// TIA Portal V18 program export: 5 tag tables, 0 data types, 0 data blocks, 6 code blocks (in call order from the OBs), 5 instance data blocks

VAR_GLOBAL   // PLC tag table "Default tag table"
   System_Byte AT %MB1 : Byte;
   FirstScan AT %M1.0 : Bool;
   DiagStatusUpdate AT %M1.1 : Bool;
   AlwaysTRUE AT %M1.2 : Bool;
   AlwaysFALSE AT %M1.3 : Bool;
   Clock_Byte AT %MB0 : Byte;
   Clock_10Hz AT %M0.0 : Bool;
   Clock_5Hz AT %M0.1 : Bool;
   "Clock_2.5Hz" AT %M0.2 : Bool;
   Clock_2Hz AT %M0.3 : Bool;
   "Clock_1.25Hz" AT %M0.4 : Bool;
   Clock_1Hz AT %M0.5 : Bool;
   "Clock_0.625Hz" AT %M0.6 : Bool;
   "Clock_0.5Hz" AT %M0.7 : Bool;
   rozlaczenie_tasmy AT %M100.2 : Bool;
   reset_licznika AT %M100.3 : Bool;
   zatrzymanie_tasmy AT %M101.2 : Bool;
   ilosc_butelek AT %MW10 : Int;
   reset_licznika_zak AT %M101.3 : Bool;
   ilosc_butelek_zak AT %MW16 : Int;
   Wylacznik_bezpieczenstwa AT %M205.0 : Bool;
   "Wlacznik/Wylacznik_glowny" AT %M206.0 : Bool;
   start_przenosik AT %M204.0 : Bool;
   stop_przenosnik AT %M204.1 : Bool;
   przenosnik_tasmowy AT %Q1.4 : Bool;
   wylacznik_przenosnika_tasmowego AT %I1.4 : Bool;
   wylacznik_nalewarki AT %I1.5 : Bool;
   wylacznik_zakrecarki AT %I1.6 : Bool;
   wylacznik_etykieciarki AT %I1.7 : Bool;
   wylacznik_pakowanie AT %I2.0 : Bool;
   samopod_start_zak AT %M102.3 : Bool;
   samopod_start_nal AT %M100.4 : Bool;
   Wlacznik_500ml AT %M207.0 : Bool;
   silownik AT %Q1.5 : Bool;
   sygnalizator_dzwiekowy AT %Q2.2 : Bool;
   robot AT %Q2.3 : Bool;
   lampa_przenosnik AT %Q2.4 : Bool;
   licznik_etykiet AT %MW50 : Int;
   cz_poj_ety AT %M210.0 : Bool;
   reset_licznika_etyk AT %M211.0 : Bool;
   pamiec_smakow AT %M100.5 : Bool;
   smak_zatrzymaj AT %M212.2 : Bool;
   czas_nalewarka AT %MD300 : Time;
   czas_pakowanie AT %MD304 : Time;
   czas_zakrecarka AT %MD308 : Time;
   cz_butelek_pakowanie AT %M230.0 : Bool;
   Tag_1 AT %MW400 : Word;
   licznik_przenosnik AT %MW30 : Int;
   res_licz_przen AT %M350.0 : Bool;
   Tag_4 AT %MD32 : Time;
   Tag_5 AT %M500.0 : Bool;
   res_licz_nalew AT %M350.1 : Bool;
   licznik_nalewarak AT %MW34 : Int;
   Tag_2 AT %M350.2 : Bool;
   Tag_3 AT %MW38 : Word;
   czas_move AT %MD312 : DWord;
   czas_w_int AT %MD316 : UDInt;
   Tag_6 AT %M320.0 : Bool;
   Tag_7 AT %MD321 : Time;
   Tag_8 AT %MD325 : Time;
   Tag_9 AT %MD329 : DInt;
   Tag_10 AT %I90.0 : Bool;
END_VAR

VAR_GLOBAL   // PLC tag table "Etykieciarka"
   start_etykieciarka AT %M102.0 : Bool;
   stop_etykieciarka AT %M102.1 : Bool;
   cz_swiatlowodowy AT %M202.0 : Bool;
   etykieta AT %Q0.6 : Bool;
   tasma_etykieciarka AT %Q0.7 : Bool;
   lampa_sygnalizacyjna_etyk AT %Q1.0 : Bool;
END_VAR

VAR_GLOBAL   // PLC tag table "Nalewarka"
   start_nalewarka AT %M100.0 : Bool;
   stop_nalewarka AT %M100.1 : Bool;
   cz_pojemnosciowy AT %M200.0 : Bool;
   dozy AT %Q0.1 : Bool;
   tasma AT %Q0.0 : Bool;
   lampa AT %Q0.2 : Bool;
   wl_pomarancza AT %M212.0 : Bool;
   pomarancza AT %Q2.5 : Bool;
   wl_truskawka AT %M212.1 : Bool;
   truskawka AT %Q2.6 : Bool;
   cz_poz_napoju AT %M213.0 : Bool;
END_VAR

VAR_GLOBAL   // PLC tag table "Pakowanie"
   start_pakowaie AT %M103.0 : Bool;
   stop_pakowanie AT %M103.1 : Bool;
   cz_pojemnosciowy_pak AT %M203.0 : Bool;
   tasma_pakowanie AT %Q1.2 : Bool;
   lampa_sygnalizacyjna_pak AT %Q1.1 : Bool;
   cz_do_robota AT %Q1.3 : Bool;
END_VAR

VAR_GLOBAL   // PLC tag table "Zakrecarka"
   start_zakrecarka AT %M101.0 : Bool;
   stop_zakrecarka AT %M101.1 : Bool;
   cz_pojemnosciowy_zak AT %M201.0 : Bool;
   tasma_zakrecarka AT %Q0.4 : Bool;
   zakretka AT %Q0.3 : Bool;
   lampa_sygnalizacyjna AT %Q0.5 : Bool;
END_VAR

ORGANIZATION_BLOCK "Main"   // OB1, LAD, ProgramCycle
TITLE = "Main Program Sweep (Cycle)"
{ S7_Optimized_Access := 'TRUE' }
VERSION : 0.1
// stored: AutoNumber true, IsIECCheckEnabled false, SetENOAutomatically false
   VAR_INPUT
      Initial_Call : Bool;   // Initial call of this OB
      Remanence : Bool;   // =True, if remanent data are available
   END_VAR
   VAR_TEMP   // added for the SCL form of the ladder/FBD networks
      _w1 : Bool;
      _w2 : Bool;
      _w3 : Bool;
      _w4 : Bool;
      _w5 : Bool;
   END_VAR
BEGIN

REGION Network 1
   // Linię produkcyjną uruchamiamy poprzez włącznik główny oraz dodatkowo każdy etap produkcji na panelu HMI.
   // Wyłącznik bezpieczeństwa znajduje się w kilku miejscach na linii produkcyjnej.
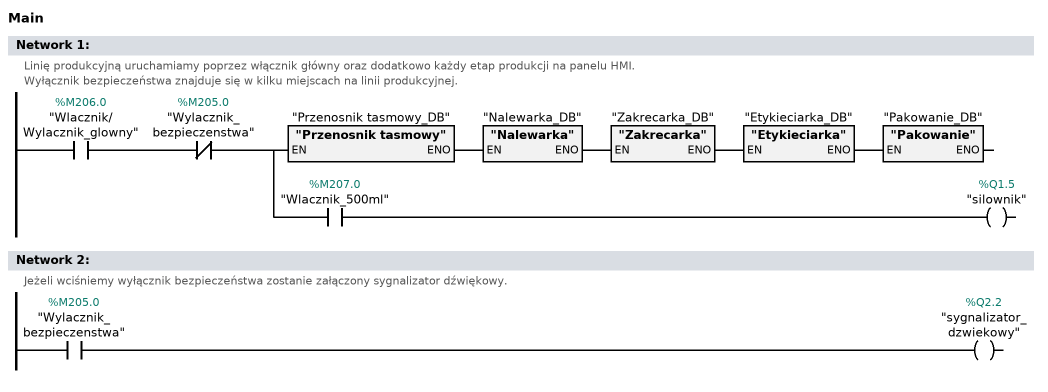
   RUNG wire#powerrail
      Contact( "Wlacznik/Wylacznik_glowny" )
      I_Contact( "Wylacznik_bezpieczenstwa" )
      wire#w1
      "Przenosnik tasmowy_DB"()
      "Nalewarka_DB"()
      "Zakrecarka_DB"()
      "Etykieciarka_DB"()
      "Pakowanie_DB"()
   END_RUNG
   RUNG wire#w1
      Contact( "Wlacznik_500ml" )
      Coil( "silownik" )
   END_RUNG
   // the same network as SCL:
   #_w1 := "Wlacznik/Wylacznik_glowny" AND NOT "Wylacznik_bezpieczenstwa";
   "Przenosnik tasmowy_DB"(EN := #_w1, ENO => #_w2);   // "Przenosnik tasmowy"
   "Nalewarka_DB"(EN := #_w2, ENO => #_w3);   // "Nalewarka"
   "Zakrecarka_DB"(EN := #_w3, ENO => #_w4);   // "Zakrecarka"
   "Etykieciarka_DB"(EN := #_w4, ENO => #_w5);   // "Etykieciarka"
   IF #_w5 THEN
       "Pakowanie_DB"();   // "Pakowanie"
   END_IF;
   "silownik" := #_w1 AND "Wlacznik_500ml";
END_REGION

REGION Network 2
   // Jeżeli wciśniemy wyłącznik bezpieczeństwa zostanie załączony sygnalizator dźwiękowy.
   RUNG wire#powerrail
      Contact( "Wylacznik_bezpieczenstwa" )
      Coil( "sygnalizator_dzwiekowy" )
   END_RUNG
   // the same network as SCL:
   "sygnalizator_dzwiekowy" := "Wylacznik_bezpieczenstwa";
END_REGION
END_ORGANIZATION_BLOCK

FUNCTION_BLOCK "Przenosnik tasmowy"   // FB5, LAD
{ S7_Optimized_Access := 'TRUE' }
VERSION : 0.1
// stored: AutoNumber true, IsIECCheckEnabled false, IsRetainMemResEnabled false, MemoryReserve 100, SetENOAutomatically false, UDAEnableTagReadback false
   VAR_TEMP
      mem0 : Time;
   END_VAR
BEGIN

REGION Network 1
   // Start przenośnika taśmowego.
   // Wyłącznik przenośnika znajduje się fizycznie na linii produkcyjnej. Stop natomiast w panelu HMI.
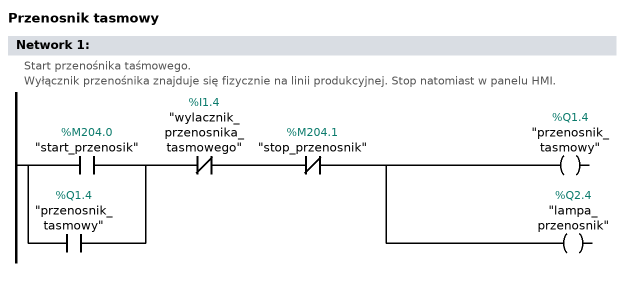
   RUNG wire#powerrail
      Contact( "start_przenosik" )
      wire#w1
      I_Contact( "wylacznik_przenosnika_tasmowego" )
      I_Contact( "stop_przenosnik" )
      wire#w2
      Coil( "przenosnik_tasmowy" )
   END_RUNG
   RUNG wire#powerrail
      Contact( "przenosnik_tasmowy" )
   END_RUNG wire#w1
   RUNG wire#w2
      Coil( "lampa_przenosnik" )
   END_RUNG
   // the same network as SCL:
   "przenosnik_tasmowy" := ("start_przenosik" OR "przenosnik_tasmowy") AND NOT "wylacznik_przenosnika_tasmowego" AND NOT "stop_przenosnik";
   "lampa_przenosnik" := "przenosnik_tasmowy";
END_REGION
END_FUNCTION_BLOCK

FUNCTION_BLOCK "Nalewarka"   // FB1, LAD
{ S7_Optimized_Access := 'TRUE' }
VERSION : 0.1
// stored: AutoNumber true, IsIECCheckEnabled false, IsRetainMemResEnabled false, MemoryReserve 100, SetENOAutomatically false, UDAEnableTagReadback false
   VAR
      czas_nalewarka : Time;
   END_VAR
   VAR_TEMP   // added for the SCL form of the ladder/FBD networks
      _w1 : Bool;
   END_VAR
BEGIN

REGION Network 1
   // Start przenośnika taśmowego i zapalenie się lampy sygnalizacyjnej.
   // Wyłącznik nalewarki znajduje się fizycznie na linii produkcyjnej, w jego skład wchodzi również system ryglowania. Stop natomiast w panelu HMI.
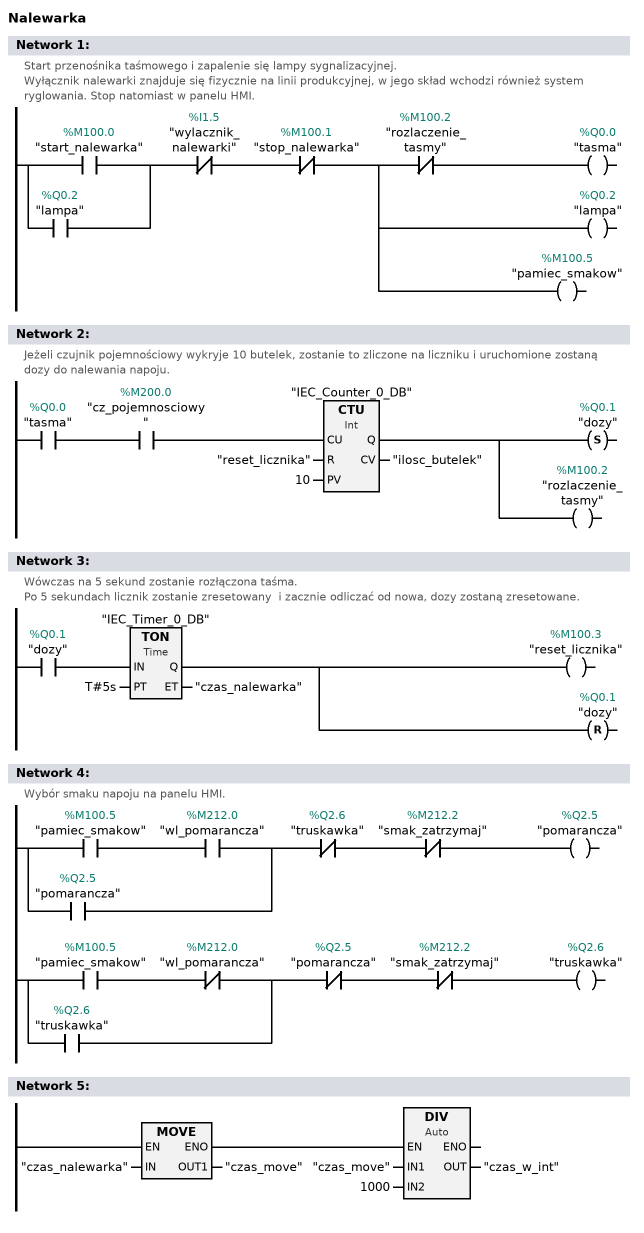
   RUNG wire#powerrail
      Contact( "start_nalewarka" )
      wire#w1
      I_Contact( "wylacznik_nalewarki" )
      I_Contact( "stop_nalewarka" )
      wire#w2
      I_Contact( "rozlaczenie_tasmy" )
      Coil( "tasma" )
   END_RUNG
   RUNG wire#powerrail
      Contact( "lampa" )
   END_RUNG wire#w1
   RUNG wire#w2
      Coil( "lampa" )
   END_RUNG
   RUNG wire#w2
      Coil( "pamiec_smakow" )
   END_RUNG
   // the same network as SCL:
   #_w1 := ("start_nalewarka" OR "lampa") AND NOT "wylacznik_nalewarki" AND NOT "stop_nalewarka";
   "tasma" := #_w1 AND NOT "rozlaczenie_tasmy";
   "lampa" := #_w1;
   "pamiec_smakow" := #_w1;
END_REGION

REGION Network 2
   // Jeżeli czujnik pojemnościowy wykryje 10 butelek, zostanie to zliczone na liczniku i uruchomione zostaną dozy do nalewania napoju.
   RUNG wire#powerrail
      Contact( "tasma" )
      Contact( "cz_pojemnosciowy" )
      { S7_Templates := "value_type := Int" } "IEC_Counter_0_DB".CTU(r := "reset_licznika", pv := 10, cv => "ilosc_butelek")
      wire#w1
      S_Coil( "dozy" )
   END_RUNG
   RUNG wire#w1
      Coil( "rozlaczenie_tasmy" )
   END_RUNG
   // the same network as SCL:
   "IEC_Counter_0_DB".CTU(CU := "tasma" AND "cz_pojemnosciowy",
                          R := "reset_licznika",
                          PV := 10,
                          CV => "ilosc_butelek");
   IF "IEC_Counter_0_DB".Q THEN "dozy" := TRUE; END_IF;
   "rozlaczenie_tasmy" := "IEC_Counter_0_DB".Q;
END_REGION

REGION Network 3
   // Wówczas na 5 sekund zostanie rozłączona taśma.
   // Po 5 sekundach licznik zostanie zresetowany  i zacznie odliczać od nowa, dozy zostaną zresetowane.
   RUNG wire#powerrail
      Contact( "dozy" )
      { S7_Templates := "time_type := Time" } "IEC_Timer_0_DB".TON(pt := T#5s, et => "czas_nalewarka")
      wire#w1
      Coil( "reset_licznika" )
   END_RUNG
   RUNG wire#w1
      R_Coil( "dozy" )
   END_RUNG
   // the same network as SCL:
   "IEC_Timer_0_DB".TON(IN := "dozy", PT := T#5s, ET => "czas_nalewarka");
   "reset_licznika" := "IEC_Timer_0_DB".Q;
   IF "IEC_Timer_0_DB".Q THEN "dozy" := FALSE; END_IF;
END_REGION

REGION Network 4
   // Wybór smaku napoju na panelu HMI.
   RUNG wire#powerrail
      Contact( "pamiec_smakow" )
      Contact( "wl_pomarancza" )
      wire#w1
      I_Contact( "truskawka" )
      I_Contact( "smak_zatrzymaj" )
      Coil( "pomarancza" )
   END_RUNG
   RUNG wire#powerrail
      Contact( "pomarancza" )
   END_RUNG wire#w1
   RUNG wire#powerrail
      Contact( "pamiec_smakow" )
      I_Contact( "wl_pomarancza" )
      wire#w2
      I_Contact( "pomarancza" )
      I_Contact( "smak_zatrzymaj" )
      Coil( "truskawka" )
   END_RUNG
   RUNG wire#powerrail
      Contact( "truskawka" )
   END_RUNG wire#w2
   // the same network as SCL:
   "pomarancza" := (("pamiec_smakow" AND "wl_pomarancza") OR "pomarancza") AND NOT "truskawka" AND NOT "smak_zatrzymaj";
   "truskawka" := (("pamiec_smakow" AND NOT "wl_pomarancza") OR "truskawka") AND NOT "pomarancza" AND NOT "smak_zatrzymaj";
END_REGION

REGION Network 5
   RUNG wire#powerrail
      Move(in := "czas_nalewarka", out1 => "czas_move")
      Div(in1 := "czas_move", in2 := 1000, out => "czas_w_int")
   END_RUNG
   // the same network as SCL:
   "czas_move" := "czas_nalewarka";
   "czas_w_int" := "czas_move" / 1000;
END_REGION
END_FUNCTION_BLOCK

FUNCTION_BLOCK "Zakrecarka"   // FB2, LAD
{ S7_Optimized_Access := 'TRUE' }
VERSION : 0.1
// stored: AutoNumber true, IsIECCheckEnabled false, IsRetainMemResEnabled false, MemoryReserve 100, SetENOAutomatically false, UDAEnableTagReadback false
   VAR_TEMP   // added for the SCL form of the ladder/FBD networks
      _w1 : Bool;
   END_VAR
BEGIN

REGION Network 1
   // Start przenośnika taśmowego i zapalenie się lampy sygnalizacyjnej.
   // Wyłącznik zakręcarki znajduje się fizycznie na linii produkcyjnej, w jego skład wchodzi również system ryglowania. Stop natomiast w panelu HMI.
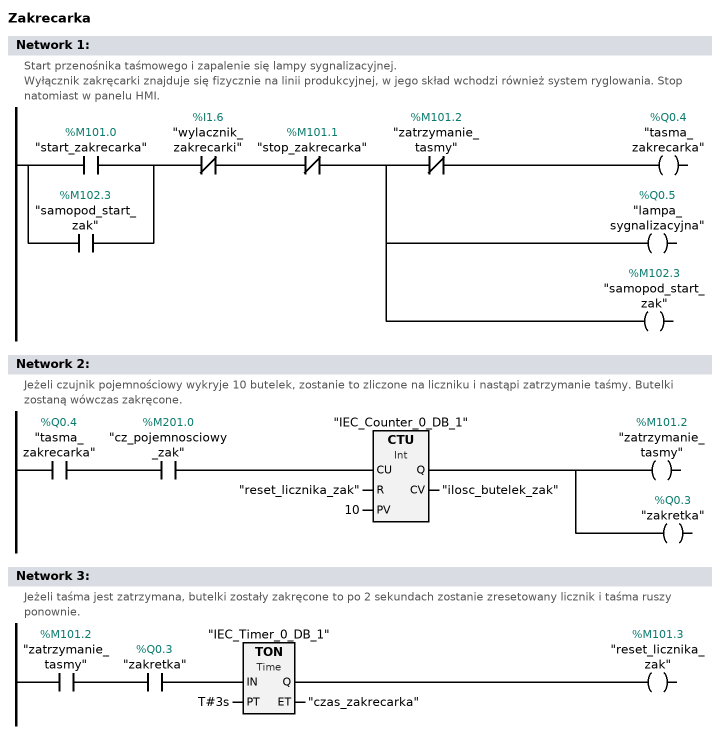
   RUNG wire#powerrail
      Contact( "start_zakrecarka" )
      wire#w1
      I_Contact( "wylacznik_zakrecarki" )
      I_Contact( "stop_zakrecarka" )
      wire#w2
      I_Contact( "zatrzymanie_tasmy" )
      Coil( "tasma_zakrecarka" )
   END_RUNG
   RUNG wire#powerrail
      Contact( "samopod_start_zak" )
   END_RUNG wire#w1
   RUNG wire#w2
      Coil( "lampa_sygnalizacyjna" )
   END_RUNG
   RUNG wire#w2
      Coil( "samopod_start_zak" )
   END_RUNG
   // the same network as SCL:
   #_w1 := ("start_zakrecarka" OR "samopod_start_zak") AND NOT "wylacznik_zakrecarki" AND NOT "stop_zakrecarka";
   "tasma_zakrecarka" := #_w1 AND NOT "zatrzymanie_tasmy";
   "lampa_sygnalizacyjna" := #_w1;
   "samopod_start_zak" := #_w1;
END_REGION

REGION Network 2
   // Jeżeli czujnik pojemnościowy wykryje 10 butelek, zostanie to zliczone na liczniku i nastąpi zatrzymanie taśmy. Butelki zostaną wówczas zakręcone.
   RUNG wire#powerrail
      Contact( "tasma_zakrecarka" )
      Contact( "cz_pojemnosciowy_zak" )
      { S7_Templates := "value_type := Int" } "IEC_Counter_0_DB_1".CTU(r := "reset_licznika_zak", pv := 10, cv => "ilosc_butelek_zak")
      wire#w1
      Coil( "zatrzymanie_tasmy" )
   END_RUNG
   RUNG wire#w1
      Coil( "zakretka" )
   END_RUNG
   // the same network as SCL:
   "IEC_Counter_0_DB_1".CTU(CU := "tasma_zakrecarka" AND "cz_pojemnosciowy_zak",
                           R := "reset_licznika_zak",
                           PV := 10,
                           CV => "ilosc_butelek_zak");
   "zatrzymanie_tasmy" := "IEC_Counter_0_DB_1".Q;
   "zakretka" := "IEC_Counter_0_DB_1".Q;
END_REGION

REGION Network 3
   // Jeżeli taśma jest zatrzymana, butelki zostały zakręcone to po 2 sekundach zostanie zresetowany licznik i taśma ruszy ponownie.
   RUNG wire#powerrail
      Contact( "zatrzymanie_tasmy" )
      Contact( "zakretka" )
      { S7_Templates := "time_type := Time" } "IEC_Timer_0_DB_1".TON(pt := T#3s, et => "czas_zakrecarka")
      Coil( "reset_licznika_zak" )
   END_RUNG
   // the same network as SCL:
   "IEC_Timer_0_DB_1".TON(IN := "zatrzymanie_tasmy" AND "zakretka", PT := T#3s, ET => "czas_zakrecarka");
   "reset_licznika_zak" := "IEC_Timer_0_DB_1".Q;
END_REGION
END_FUNCTION_BLOCK

FUNCTION_BLOCK "Etykieciarka"   // FB3, LAD
{ S7_Optimized_Access := 'TRUE' }
VERSION : 0.1
// stored: AutoNumber true, IsIECCheckEnabled false, IsRetainMemResEnabled false, MemoryReserve 100, SetENOAutomatically false, UDAEnableTagReadback false
BEGIN

REGION Network 1
   // Start przenośnika taśmowego i zapalenie się lampy sygnalizacyjnej.
   // Wyłącznik etykieciarki znajduje się fizycznie na linii produkcyjnej. Stop natomiast w panelu HMI.
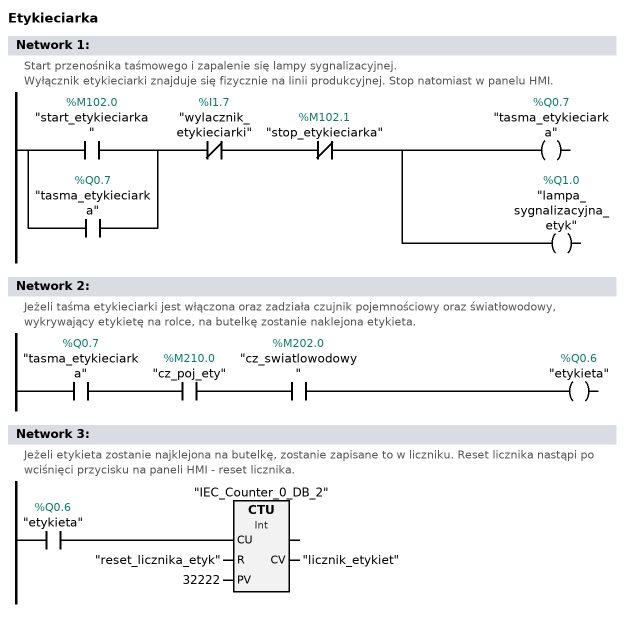
   RUNG wire#powerrail
      Contact( "start_etykieciarka" )
      wire#w1
      I_Contact( "wylacznik_etykieciarki" )
      I_Contact( "stop_etykieciarka" )
      wire#w2
      Coil( "tasma_etykieciarka" )
   END_RUNG
   RUNG wire#powerrail
      Contact( "tasma_etykieciarka" )
   END_RUNG wire#w1
   RUNG wire#w2
      Coil( "lampa_sygnalizacyjna_etyk" )
   END_RUNG
   // the same network as SCL:
   "tasma_etykieciarka" := ("start_etykieciarka" OR "tasma_etykieciarka") AND NOT "wylacznik_etykieciarki" AND NOT "stop_etykieciarka";
   "lampa_sygnalizacyjna_etyk" := "tasma_etykieciarka";
END_REGION

REGION Network 2
   // Jeżeli taśma etykieciarki jest włączona oraz zadziała czujnik pojemnościowy oraz światłowodowy, wykrywający etykietę na rolce, na butelkę zostanie naklejona etykieta.
   RUNG wire#powerrail
      Contact( "tasma_etykieciarka" )
      Contact( "cz_poj_ety" )
      Contact( "cz_swiatlowodowy" )
      Coil( "etykieta" )
   END_RUNG
   // the same network as SCL:
   "etykieta" := "tasma_etykieciarka" AND "cz_poj_ety" AND "cz_swiatlowodowy";
END_REGION

REGION Network 3
   // Jeżeli etykieta zostanie najklejona na butelkę, zostanie zapisane to w liczniku. Reset licznika nastąpi po wciśnięci przycisku na paneli HMI - reset licznika.
   RUNG wire#powerrail
      Contact( "etykieta" )
      { S7_Templates := "value_type := Int" } "IEC_Counter_0_DB_2".CTU(r := "reset_licznika_etyk", pv := 32222, cv => "licznik_etykiet")
   END_RUNG
   // the same network as SCL:
   "IEC_Counter_0_DB_2".CTU(CU := "etykieta", R := "reset_licznika_etyk", PV := 32222, CV => "licznik_etykiet");
END_REGION
END_FUNCTION_BLOCK

FUNCTION_BLOCK "Pakowanie"   // FB4, LAD
{ S7_Optimized_Access := 'TRUE' }
VERSION : 0.1
// stored: AutoNumber true, IsIECCheckEnabled false, IsRetainMemResEnabled false, MemoryReserve 100, SetENOAutomatically false, UDAEnableTagReadback false
BEGIN

REGION Network 1
   // Start przenośnika taśmowego i zapalenie się lampy sygnalizacyjnej.
   // Wyłącznik pakowania znajduje się fizycznie na linii produkcyjnej, w jego skład wchodzi również kurtyna świetlna. Stop natomiast w panelu HMI.
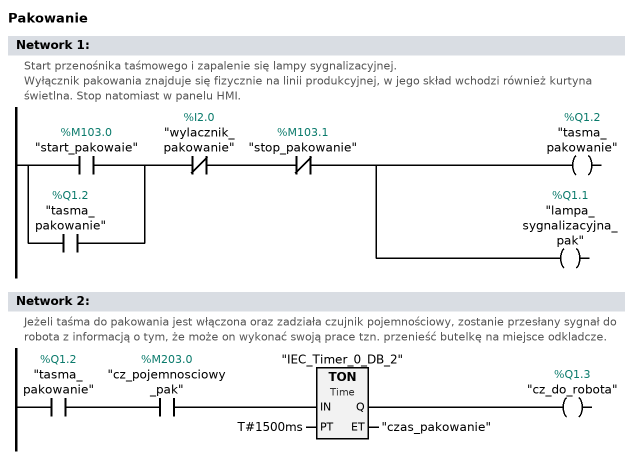
   RUNG wire#powerrail
      Contact( "start_pakowaie" )
      wire#w1
      I_Contact( "wylacznik_pakowanie" )
      I_Contact( "stop_pakowanie" )
      wire#w2
      Coil( "tasma_pakowanie" )
   END_RUNG
   RUNG wire#powerrail
      Contact( "tasma_pakowanie" )
   END_RUNG wire#w1
   RUNG wire#w2
      Coil( "lampa_sygnalizacyjna_pak" )
   END_RUNG
   // the same network as SCL:
   "tasma_pakowanie" := ("start_pakowaie" OR "tasma_pakowanie") AND NOT "wylacznik_pakowanie" AND NOT "stop_pakowanie";
   "lampa_sygnalizacyjna_pak" := "tasma_pakowanie";
END_REGION

REGION Network 2
   // Jeżeli taśma do pakowania jest włączona oraz zadziała czujnik pojemnościowy, zostanie przesłany sygnał do robota z informacją o tym, że może on wykonać swoją prace tzn. przenieść butelkę na miejsce odkladcze.
   RUNG wire#powerrail
      Contact( "tasma_pakowanie" )
      Contact( "cz_pojemnosciowy_pak" )
      { S7_Templates := "time_type := Time" } "IEC_Timer_0_DB_2".TON(pt := T#1500ms, et => "czas_pakowanie")
      Coil( "cz_do_robota" )
   END_RUNG
   // the same network as SCL:
   "IEC_Timer_0_DB_2".TON(IN := "tasma_pakowanie" AND "cz_pojemnosciowy_pak",
                          PT := T#1500ms,
                          ET => "czas_pakowanie");
   "cz_do_robota" := "IEC_Timer_0_DB_2".Q;
END_REGION
END_FUNCTION_BLOCK

DATA_BLOCK "Etykieciarka_DB"   // DB7
VERSION : 0.1
// stored: AutoNumber true, DBAccessibleFromOPCUA true, DBAccessibleFromWebserver true, InstanceOfName Etykieciarka, InstanceOfType FB
"Etykieciarka"
BEGIN
END_DATA_BLOCK

DATA_BLOCK "Nalewarka_DB"   // DB3
VERSION : 0.1
// stored: AutoNumber true, DBAccessibleFromOPCUA true, DBAccessibleFromWebserver true, InstanceOfName Nalewarka, InstanceOfType FB
"Nalewarka"
BEGIN
END_DATA_BLOCK

DATA_BLOCK "Pakowanie_DB"   // DB9
VERSION : 0.1
// stored: AutoNumber true, DBAccessibleFromOPCUA true, DBAccessibleFromWebserver true, InstanceOfName Pakowanie, InstanceOfType FB
"Pakowanie"
BEGIN
END_DATA_BLOCK

DATA_BLOCK "Przenosnik tasmowy_DB"   // DB12
VERSION : 0.1
// stored: AutoNumber true, DBAccessibleFromOPCUA true, DBAccessibleFromWebserver true, InstanceOfName Przenosnik tasmowy, InstanceOfType FB
"Przenosnik tasmowy"
BEGIN
END_DATA_BLOCK

DATA_BLOCK "Zakrecarka_DB"   // DB6
VERSION : 0.1
// stored: AutoNumber true, DBAccessibleFromOPCUA true, DBAccessibleFromWebserver true, InstanceOfName Zakrecarka, InstanceOfType FB
"Zakrecarka"
BEGIN
END_DATA_BLOCK
